(* IEC 61131-3 sources: CodesysTest/export/ObjectHandling/FB_CollectionHandlerHomable.pou, 2 files *)

(* ---- FB_CollectionHandlerHomable.pou.st ---- *)
(*#-#-#-#-#-#-#-#-#-#---Declaration---#-#-#-#-#-#-#-#-#-#-#-#-#*)

FUNCTION_BLOCK FB_CollectionHandlerHomable
VAR_INPUT

END_VAR
VAR
	Collection: ARRAY[0..GlobalObjects.MAX_LOGGABLE] OF IInitializable; // object array
	ObjNames   : ARRAY[0..GlobalObjects.MAX_LOGGABLE] OF STRING;
	_ArrayOver   : BOOL;
	_BadObj      : INT;
	_DupeObj   : INT;
	_OverObj   : INT;
	_TotalObj   : UINT;
END_VAR(*#-#-#-#-#-#-#-#-#-#---Implementation---#-#-#-#-#-#-#-#-#-#-#-#-#*)

//	Function Block: FB_CollectionHandlerLoggable
//	Description: This collection handler takes in loggable objects and registers them with a logger.  The FirstScan function should trigger the
//				 RegisterAll() method to register all loggable objects with a logger
//	Created by: Ben Hess
//	Created Date: Tuesday, September 11, 2018

(* ---- HomeAll.m.st ---- *)
(*#-#-#-#-#-#-#-#-#-#---Declaration---#-#-#-#-#-#-#-#-#-#-#-#-#*)

METHOD HomeAll
VAR_INPUT

END_VAR
VAR
	J : UINT;
	Cast : IHomable;
END_VAR
(*#-#-#-#-#-#-#-#-#-#---Implementation---#-#-#-#-#-#-#-#-#-#-#-#-#*)

FOR J:= 0 TO _TotalObj - 1 DO
	IF (__QUERYINTERFACE(Collection[J], Cast)) THEN
		Cast.HomeNow();
	ELSE
		RETURN;
	END_IF
END_FOR
